(*

.. <legal notes>

legal notes
=================
| SPDX-FileCopyrightText: © 2025 Oleksandr Tiutyk <trofimich@gmail.com>
| SPDX-License-Identifier: LGPL-3.0-only
| For details check: LGPL-3.0-only_

.. _LGPL-3.0-only: https://www.gnu.org/licenses/lgpl-3.0.en.html

.. </legal notes>

*)

INTERFACE IComparable EXTENDS __System.IQueryInterface

METHOD ComapreTo : COMPARISION_RESULT
VAR_IN_OUT CONSTANT
	otherValue : IComparable;
END_VAR
END_METHOD

END_INTERFACE

(* stored: Version 1.1.0.1
   Itf IComparable: Id {f57543d2-c48b-40a1-89a1-48969e8514ee}
   Method ComapreTo: Id {2475bd0e-54ae-4479-a8b3-6f2c5ca19e19} *)
